{attribute 'GeneratedUsingTerminal: EL3311-0000-0018'}
{attribute addProperty BoxType "EL3311-0000-0018"}
{attribute addProperty Id "StatusAT %I*Status_F2CE6D917ValueAT %I*INT2"}
{attribute addProperty CRC "1245267073"}
{attribute addProperty Size "9"}
TYPE TC_Inputs_4A394481 :
STRUCT
	{attribute addProperty Name "Status"}
	Status AT %I* : Status_F2CE6D91;
	{attribute addProperty Name "Value"}
	Value AT %I* : INT;
END_STRUCT
END_TYPE

(* stored: Version 1.2.0.0, ProductVersion 3.1.4024.9
   DUT TC_Inputs_4A394481: Id {e43f438e-8789-4e7f-923b-a41cee0d342f} *)
